FUNCTION_BLOCK FB_TrafficLightHandler
VAR_INPUT
END_VAR
VAR_OUTPUT
END_VAR
VAR
	
Lights : ST_TrafficLight;

END_VAR

{attribute 'TcRpcEnable'}
METHOD M_RequestAllLightOff : BOOL
VAR_INPUT
END_VAR
Lights.GreenLight :=FALSE;
Lights.YellowLight := FALSE;
Lights.RedLight := FALSE;
END_METHOD

{attribute 'TcRpcEnable'}
METHOD M_RequestAllLightOn : BOOL
VAR_INPUT
END_VAR
Lights.GreenLight := TRUE;
Lights.YellowLight := TRUE;
Lights.RedLight := TRUE;
END_METHOD

END_FUNCTION_BLOCK

(* stored: Version 1.1.0.1, ProductVersion 3.1.4024.11
   POU FB_TrafficLightHandler: Id {f67fd037-6f4e-4130-9d91-159c673bd474}, SpecialFunc None
   Method M_RequestAllLightOff: Id {fe5063b3-e218-470d-8cde-843d02c1d4d0}
   Method M_RequestAllLightOn: Id {367ddf6f-94d7-4eb6-94fc-4d7629ee7b7b} *)
